//==================================================================================================
//							Beckhoff Automation Poland
//							FB_TaskInfo
//							15.11.2016
//
//				Blok funkcyjny odczytujący informacje o tasku
//				Zapamiętuje maksymalne czasy wykonania oraz licznik przekroczeń
//
// 	v1.1 	|| TC v 3.1.4020.14 	|| - dodanie wyjsc
// 	v1.0 	|| TC v 3.1.4020.14 	|| - pierwsza wersja
//==================================================================================================
FUNCTION_BLOCK FB_TaskInfo
VAR_INPUT
	bReset					: BOOL;
END_VAR
VAR_OUTPUT
	bError					: BOOL;
END_VAR
VAR
	fbGetCurTaskIdx			: GETCURTASKINDEX;
	rLastExecTime			: REAL;
	rCycleTime				: REAL;
	uiPriority				: UINT;
	sTaskName				: STRING(63);
	bCycleTimeExceeded		: BOOL;
	rCycleCount				: REAL;
	rTotalTime				: REAL;
	rAverageCycleTime		: REAL;
	bResetVisu				: BOOL;
	byIndex					: BYTE;
END_VAR
VAR PERSISTENT
	udiCountExceedCycle		: UDINT; 						
	rMaxExecTime			: REAL;						
END_VAR

fbGetCurTaskIdx(index=>byIndex);

(*Odczyt czasu cyklu i ostatniego czasu wykonania*)
rCycleTime 					:= UDINT_TO_REAL(_TaskInfo[byIndex].CycleTime)/10000.0;
rLastExecTime 				:= UDINT_TO_REAL(_TaskInfo[byIndex].LastExecTime)/10000.0;
(*Zapamiętanie maksymalnego czasu wykonania*)
IF rLastExecTime > rMaxExecTime THEN 
	rMaxExecTime 			:= rLastExecTime;
END_IF

uiPriority					:= _TaskInfo[byIndex].Priority;
sTaskName					:= _TaskInfo[byIndex].TaskName;
bCycleTimeExceeded			:= _TaskInfo[byIndex].CycleTimeExceeded;
bError 						:= bCycleTimeExceeded; // Blad gdy czas cyklu przekroczony

(*Licznik przekroczeń czasu cyklu*)
IF _TaskInfo[byIndex].CycleTimeExceeded  THEN 
	udiCountExceedCycle 	:= udiCountExceedCycle + 1; 
END_IF
rCycleCount 				:= rCycleCount + 1;
rTotalTime 					:= rLastExecTime + rTotalTime;
rAverageCycleTime 			:= rTotalTime / rCycleCount;

(*Reset wyliczanych wartości*)
IF bReset OR bResetVisu THEN
	udiCountExceedCycle 	:= 0;
	rMaxExecTime 			:= 0;
	rTotalTime 				:= 0;
	rCycleCount 			:= 0;
	rAverageCycleTime 		:= 0;
	bReset 					:= FALSE;
END_IF

END_FUNCTION_BLOCK

(* stored: Version 1.1.0.1, ProductVersion 3.1.4026.13, FileIdentifier 56e23694a30a0a8c8f90c2faaf6206ecdfe2e041, FileSignature 337c429bf80461d6631ae364acd770fec3625d08afdc2f859806e42a2cee5664154530440bb43afe1a90f97af6e79d7193fa1067dc1639fa74a91004e1c9c9499543077f354e228761d1ea8bc53997e0f99881c6451b98a0b6dbaaf0a99e7807d5a0f886036e81e02e289a26a307a83ca277cc8c4b7d5b5342cd9a66f25678c610faf898b2bcfaeb993f6aa81a53ee2219a6e4784661f9014a8e5b7df570bbafc9dcad05170d34544e3d400f2e291dc1a5e17d7af7d3a98f9e4f88a2240d8d44762772ef143b808656467d38ab73a874fb8548e0f7f95ecb9ec94dd1024c23e658ec2947f4064c9e74c68d9696360e41b14d0012b6ffa99cb02b53b3e55b90d7
   POU FB_TaskInfo: Id {a97cad04-5914-49fc-bdc9-2d2ccb5425d6}, SpecialFunc None *)
